(* IEC 61131-3 sources: br_struct_parser/a51/BR_sample_task, 3 files *)

(* ---- Types.typ ---- *)
TYPE
	testStruct_typ : 	STRUCT
		New_Member6 : UDINT := 1;
		New_Member5 : USINT := 25;
		New_Member7 : SINT := -5;
		New_Member1 : USINT := 5;
		New_Member2 : UINT := 18;
		New_Member3 : testSubstructTyp;
		New_Member4 : STRING[80] := 'hallowelt';
	END_STRUCT;
	testSubstructTyp : 	STRUCT
		New_Member2 : DATE_AND_TIME;
		New_Member3 : USINT := 255;
		New_Member1 : UDINT := 455667;
	END_STRUCT;
END_TYPE

(* ---- Main.st ---- *)
PROGRAM _INIT
	(* Insert code here *)

END_PROGRAM

PROGRAM _CYCLIC

	teststruct;

	CASE step OF
		0: // warte
			FileDelete_0.enable:=0;
			FileCreate_0.enable:=0;
			FileWrite_0.enable:=0;
			FileClose_0.enable:=0;

		1: //löschen alte datei
			IF FileDelete_0.enable=0 THEN
				FileDelete_0.enable := 1;
				FileDelete_0.pDevice:=ADR(LOCALDEVICE);
				FileDelete_0.pName:=ADR('web/a51/myStruct.bin');
			END_IF;
			IF FileDelete_0.status  <> ERR_FUB_BUSY AND FileDelete_0.status <> ERR_FUB_ENABLE_FALSE THEN
				FileDelete_0.enable:=0;
				step:=2;
			END_IF;

		2: //create neue
			IF FileCreate_0.enable=0 THEN
				FileCreate_0.enable := 1;
				FileCreate_0.pDevice:=ADR(LOCALDEVICE);
				FileCreate_0.pFile:=ADR('web/a51/myStruct.bin');
			END_IF;

			IF FileCreate_0.status  <> ERR_FUB_BUSY AND FileCreate_0.status  <> ERR_FUB_ENABLE_FALSE THEN
				FileCreate_0.enable:=0;
				IF FileCreate_0.status <> ERR_OK THEN
					step:=0;
				ELSE
					step:=3;
					fileIdent:=FileCreate_0.ident;
				END_IF;
			END_IF;

		3:// schreiben

			IF FileWrite_0.enable=0 THEN
				FileWrite_0.ident:=fileIdent;
				FileWrite_0.offset:=0;
				FileWrite_0.pSrc:=ADR(teststruct);
				FileWrite_0.len:=SIZEOF(teststruct);
				FileWrite_0.enable:=1;
			END_IF;
			IF FileWrite_0.status  <> ERR_FUB_BUSY AND FileWrite_0.status  <> ERR_FUB_ENABLE_FALSE THEN
				FileWrite_0.enable:=0;
				IF FileWrite_0.status <> ERR_OK THEN
					step:=0;
				ELSE
					step:=4;

				END_IF;
			END_IF;
		4://schließen

			IF FileClose_0.enable=0 THEN
				FileClose_0.ident:=fileIdent;
				FileClose_0.enable:=1;
			END_IF;
			IF FileClose_0.status  <> ERR_FUB_BUSY AND FileClose_0.status  <> ERR_FUB_ENABLE_FALSE THEN
				FileClose_0.enable:=0;
				step:=0;
			END_IF;
	END_CASE;

	FileDelete_0();
	FileCreate_0();
	FileWrite_0();
	FileClose_0();

END_PROGRAM

PROGRAM _EXIT
	(* Insert code here *)

END_PROGRAM

(* ---- Variables.var ---- *)
VAR
	teststruct : testStruct_typ;
	fileIdent : UDINT;
	offsetStruct : UDINT;
	size : UDINT;
	lenStruct : UDINT;
	FileClose_0 : FileClose;
	FileWrite_0 : FileWrite;
	FileCreate_0 : FileCreate;
	FileDelete_0 : FileDelete;
	step : USINT;
END_VAR
